FUNCTION F_SetSBPumpStatuses : BOOL
VAR_INPUT
	stExpStatus : ST_SBPumpStatuses;
END_VAR
VAR
END_VAR

GVL_BTS_VAC.fb_PP_PMF.M_Run(stExpStatus.bRoughingPumpOn); 
GVL_BTS_VAC.fb_PP_PTM.M_Run(stExpStatus.bTurboPumpOn);
GVL_BTS_VAC.fb_PP_PIP.M_Run(stExpStatus.bIonPumpOn);

END_FUNCTION

(* stored: Version 1.1.0.1, ProductVersion 3.1.4022.17
   POU F_SetSBPumpStatuses: Id {b84ef4b3-32da-49d5-b9da-dd56cc2c945f}, SpecialFunc None *)
